{attribute addProperty BoxType "AT2020-0250-0023"}
{attribute addProperty Id "A_0073_AT2000_5250_0016_AT2000_5250AT2000_3DCFC8D064080"}
{attribute addProperty CRC "2564417865"}
{attribute addProperty SizeInBites "640"}
{attribute addProperty SizeInBytes "80"}
TYPE A_0061_AT2020_0250_0023_AT2020_0250_98D9E949 EXTENDS AT2020_9506A482 :
STRUCT
	{attribute addProperty Name "A_0073_AT2000_5250_0016_AT2000_5250"}
	A_0073_AT2000_5250_0016_AT2000_5250 : AT2000_3DCFC8D0;
END_STRUCT
END_TYPE

(* stored: Version 1.2.0.0, ProductVersion 3.1.4024.9
   DUT A_0061_AT2020_0250_0023_AT2020_0250_98D9E949: Id {a8521cac-a27e-44d2-97f0-031d810f4b9b} *)
